// TIA Portal V19 export
FUNCTION "STOP PRESTERIL" : Void   // FC45, STL
TITLE = STOP PRESTERILIZING TANK
{ S7_Optimized_Access := 'TRUE' }
NAME : SPRESTE
VERSION : 0.0
// Comment
// stored: AutoNumber false
BEGIN

NETWORK
TITLE = STOP PRESTERILIZING TANK
// Comment
      A     "S0 STOP PRESTE. TANK";
      JC    M001;
      R     "S1 STOP PRESTE. TANK";
      R     "S2 STOP PRESTE. TANK";
      BEU;
M001: A     "S1 STOP PRESTE. TANK";
      JC    M002;
      R     "MY0545";
      R     "MY0148";
      R     "MY0103";
      R     "MY0104";
      R     "MY0143";
      R     "MY0112";
      R     "MY0113";
      R     "MY0147";
      R     "MY0144";
      R     "MY0136";
      R     "MY0135";
      R     "MY0137";
      R     "MY0124";
      R     "MY0111";
      R     "IF_Device".V_09_30.IO.V._IO.IN.Activate;
      R     "IF_Device".V_09_31.IO.V._IO.IN.Activate;
      R     "PULSE 01.18 PRESTERILI";
      R     "SPIN 01.30 PRESTERILI";
      R     "TEST TEMPS. PRESTERILI";
      R     "TEST BARRIERS";
      R     "T 14 STERILE TIME";
      R     "T 15 COOLING TIME";
      R     "AutoPT0167/IP0149";
      R     "T 16 BLOW OUT COND";
//     R     "MM01.30"
      R     "TANK STERILE";
      R     "ManPT0167/IP0149";
      R     "TEST FILLING PRESSURE";
      S     "S1 STOP PRESTE. TANK";
//;
      R     "MY0901";
      R     "MY0904";
      R     "MY0906";
      R     "MY0907";
      R     "M_Barrier_Sterile";
      R     "M_Barrier_Sterlising";
//;
      BEU;
M002: NOP   0;

NETWORK
TITLE = 
// Comment
      A     "S2 STOP PRESTE. TANK";
      JC    c001;
      L     "MeasuredValues".TT0176REAL;  //"DB-ANALOG INPUT".TT0176MEAS
      L     "Setpoints".TT0176MaxTotalStop;  //"DB SETPOINTS".TT0176MaxTotalStop
      <R;
      R     "S0 STOP PRESTE. TANK";
      BEC;
      S     "MY0109";
      S     "TIM15";
      S     "S2 STOP PRESTE. TANK";
      BEU;
c001: NOP   0;

NETWORK
TITLE = 
// WAIT FOR COOLING TIMER.
// IF THE PRESSURE IN THE STERILE TANK FALL BELOW MINIMUM PRESSURE, 
// THEN OPEN TO DRAIN TO AVOID VACUUM (COLLAPS) IN TANK.
// THIS VACUUM COULD OCCUR IF COOLING HAPPENS FAST.
      A     "S3 STOP PRESTE. TANK";
      JC    c002;
      AN    "T 15 COOLING TIME";
      R     "S0 STOP PRESTE. TANK";
      BEC;
      L     "MeasuredValues".PT0167REAL;  // "DB-ANALOG INPUT".PT0167MeasPressure
      L     "Setpoints".PresForOpenDrain;  //"DB SETPOINTS".PresForOpenDrain
      >R;  // OPEN TO DRAIN IF PRESSURE TOO LOW
      BEC;
      S     "MY0112";
      S     "MY0113";
      S     "MY0114";
      S     "MY0111";
      BEU;
c002: NOP   0;
END_FUNCTION
